{attribute addProperty BoxType "EP4378-1022-0017"}
{attribute addProperty Id "OutputAT %Q*BOOL81"}
{attribute addProperty CRC "2134331056"}
{attribute addProperty SizeInBites "8"}
{attribute addProperty SizeInBytes "1"}
TYPE DO_X08_Pin4_Output_7F374EB0 :
STRUCT
	{attribute addProperty Name "Output"}
	Output AT %Q* : BOOL;
END_STRUCT
END_TYPE

(* stored: Version 1.2.0.0, ProductVersion 3.1.4024.9
   DUT DO_X08_Pin4_Output_7F374EB0: Id {ddbd925b-6b0e-4a85-8acb-4deae2a8122a} *)
